FUNCTION_BLOCK FB_Car EXTENDS FB_Vehicle


VAR_IN_OUT
	fbEngine : FB_PetrolEngine;
END_VAR
VAR
	fCurrentFuelLimit : REAL := 42342423;
END_VAR


IF bMoving THEN
	fCurrentFuelLimit := fCurrentFuelLimit - 20;
END_IF

METHOD Feuling : BOOL
VAR_INPUT
END_VAR
bMoving := FALSE;
fCurrentFuelLimit := fFuelKilometerLimit;
END_METHOD

END_FUNCTION_BLOCK

(* stored: Version 1.1.0.1, ProductVersion 3.1.4024.16
   POU FB_Car: Id {64f4a3f7-7bc8-4255-8be5-c373cd978fbd}, SpecialFunc None
   Method Feuling: Id {74b70f8e-f221-4924-bec1-697fe9a436c5} *)
